// Mitsubishi GX Works2 project: hello   PLC: Q03UDV

PROGRAM MAIN
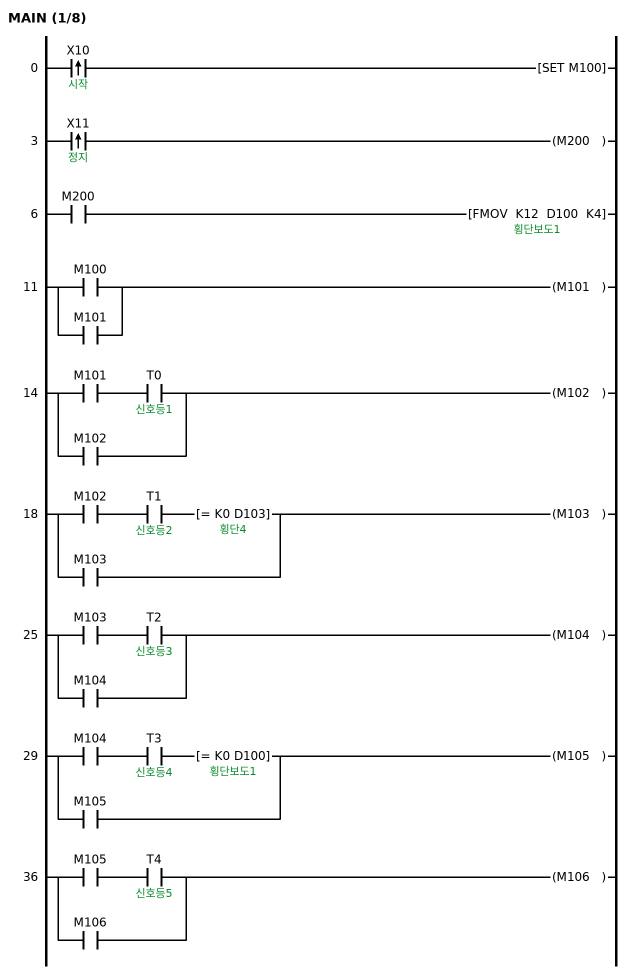
0     LDP     X10  ; 시작
      SET     M100
3     LDP     X11  ; 정지
      OUT     M200
6     LD      M200
      FMOV    K12 D100 K4  ; 횡단보도1
11    LD      M100
      OR      M101
      OUT     M101
14    LD      M101
      AND     T0  ; 신호등1
      OR      M102
      OUT     M102
18    LD      M102
      AND     T1  ; 신호등2
      AND=    K0 D103  ; 횡단4
      OR      M103
      OUT     M103
25    LD      M103
      AND     T2  ; 신호등3
      OR      M104
      OUT     M104
29    LD      M104
      AND     T3  ; 신호등4
      AND=    K0 D100  ; 횡단보도1
      OR      M105
      OUT     M105
36    LD      M105
      AND     T4  ; 신호등5
      OR      M106
      OUT     M106
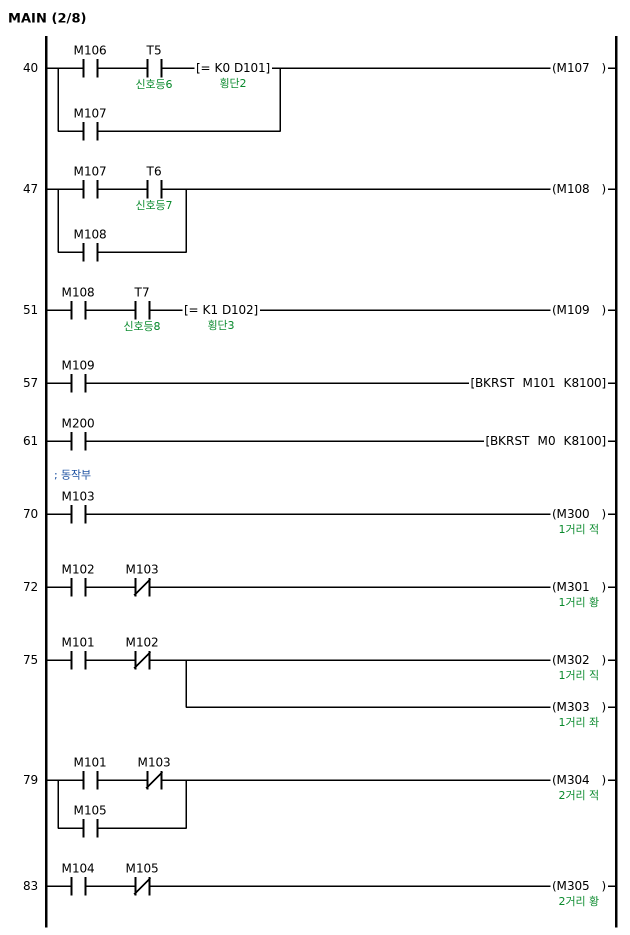
40    LD      M106
      AND     T5  ; 신호등6
      AND=    K0 D101  ; 횡단2
      OR      M107
      OUT     M107
47    LD      M107
      AND     T6  ; 신호등7
      OR      M108
      OUT     M108
51    LD      M108
      AND     T7  ; 신호등8
      AND=    K1 D102  ; 횡단3
      OUT     M109
57    LD      M109
      BKRST   M101 K8100
61    LD      M200
      BKRST   M0 K8100
; 동작부
70    LD      M103
      OUT     M300  ; 1거리 적
72    LD      M102
      ANI     M103
      OUT     M301  ; 1거리 황
75    LD      M101
      ANI     M102
      OUT     M302  ; 1거리 직
      OUT     M303  ; 1거리 좌
79    LD      M101
      ANI     M103
      OR      M105
      OUT     M304  ; 2거리 적
83    LD      M104
      ANI     M105
      OUT     M305  ; 2거리 황
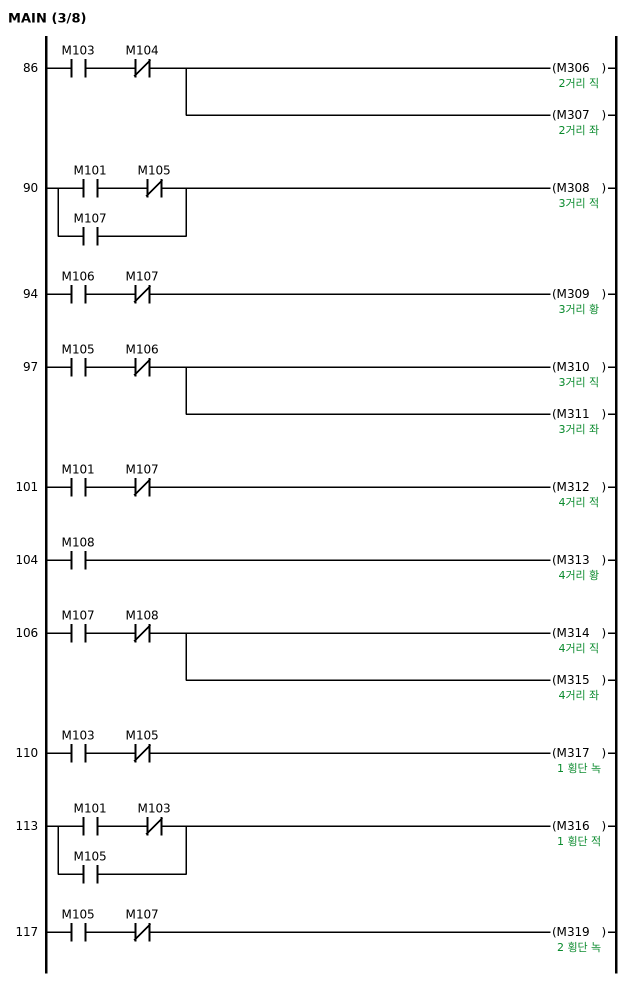
86    LD      M103
      ANI     M104
      OUT     M306  ; 2거리 직
      OUT     M307  ; 2거리 좌
90    LD      M101
      ANI     M105
      OR      M107
      OUT     M308  ; 3거리 적
94    LD      M106
      ANI     M107
      OUT     M309  ; 3거리 황
97    LD      M105
      ANI     M106
      OUT     M310  ; 3거리 직
      OUT     M311  ; 3거리 좌
101   LD      M101
      ANI     M107
      OUT     M312  ; 4거리 적
104   LD      M108
      OUT     M313  ; 4거리 황
106   LD      M107
      ANI     M108
      OUT     M314  ; 4거리 직
      OUT     M315  ; 4거리 좌
110   LD      M103
      ANI     M105
      OUT     M317  ; 1 횡단 녹
113   LD      M101
      ANI     M103
      OR      M105
      OUT     M316  ; 1 횡단 적
117   LD      M105
      ANI     M107
      OUT     M319  ; 2 횡단 녹
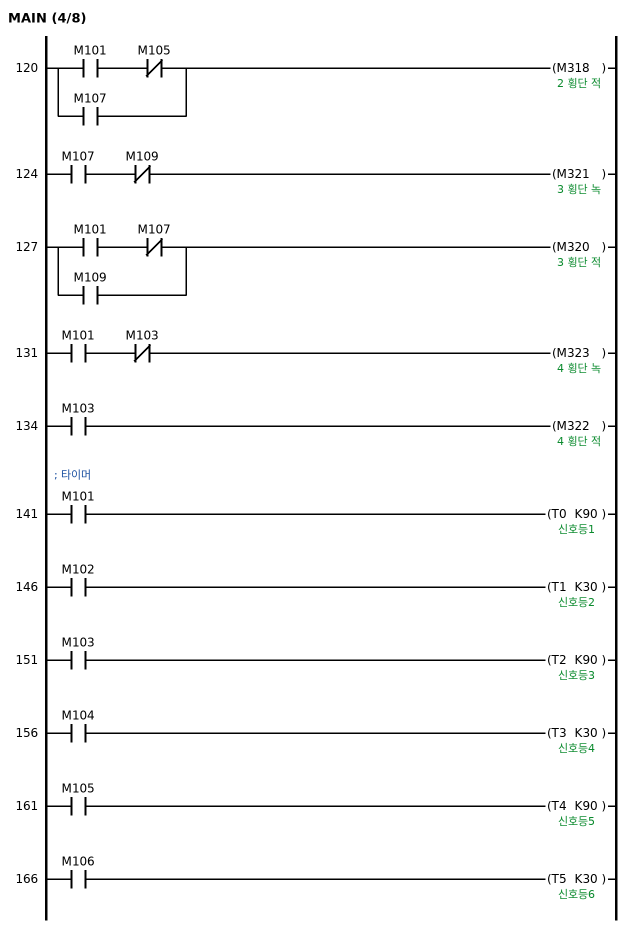
120   LD      M101
      ANI     M105
      OR      M107
      OUT     M318  ; 2 횡단 적
124   LD      M107
      ANI     M109
      OUT     M321  ; 3 횡단 녹
127   LD      M101
      ANI     M107
      OR      M109
      OUT     M320  ; 3 횡단 적
131   LD      M101
      ANI     M103
      OUT     M323  ; 4 횡단 녹
134   LD      M103
      OUT     M322  ; 4 횡단 적
; 타이머
141   LD      M101
      OUT     T0 K90  ; 신호등1
146   LD      M102
      OUT     T1 K30  ; 신호등2
151   LD      M103
      OUT     T2 K90  ; 신호등3
156   LD      M104
      OUT     T3 K30  ; 신호등4
161   LD      M105
      OUT     T4 K90  ; 신호등5
166   LD      M106
      OUT     T5 K30  ; 신호등6
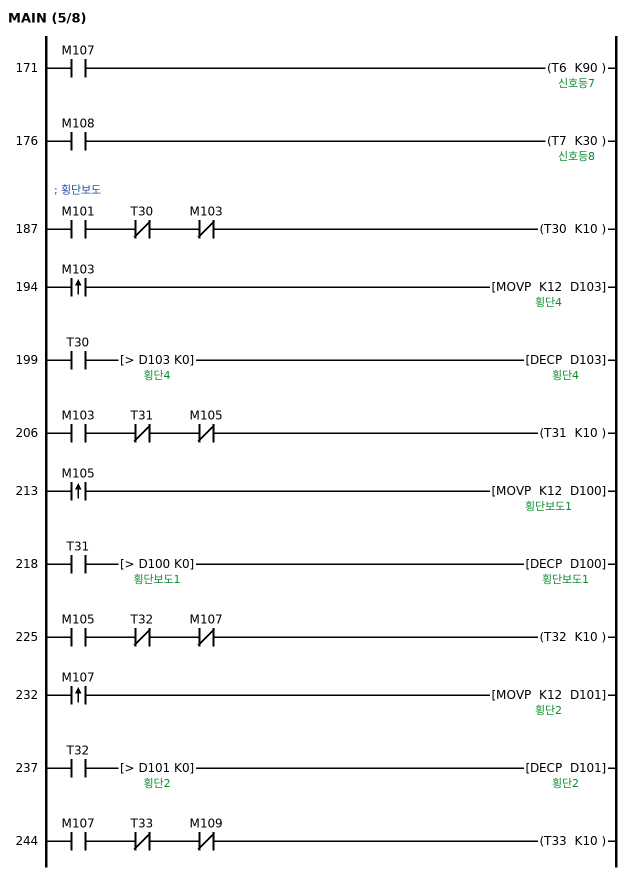
171   LD      M107
      OUT     T6 K90  ; 신호등7
176   LD      M108
      OUT     T7 K30  ; 신호등8
; 횡단보도
187   LD      M101
      ANI     T30
      ANI     M103
      OUT     T30 K10
194   LDP     M103
      MOVP    K12 D103
199   LD      T30
      AND>    D103 K0  ; 횡단4
      DECP    D103
206   LD      M103
      ANI     T31
      ANI     M105
      OUT     T31 K10
213   LDP     M105
      MOVP    K12 D100
218   LD      T31
      AND>    D100 K0  ; 횡단보도1
      DECP    D100
225   LD      M105
      ANI     T32
      ANI     M107
      OUT     T32 K10
232   LDP     M107
      MOVP    K12 D101
237   LD      T32
      AND>    D101 K0  ; 횡단2
      DECP    D101
244   LD      M107
      ANI     T33
      ANI     M109
      OUT     T33 K10
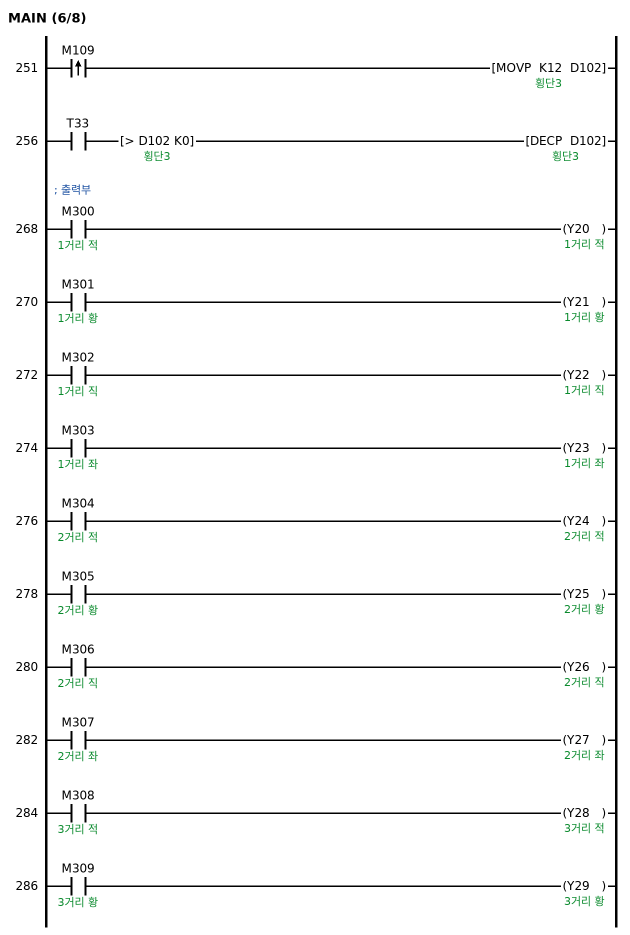
251   LDP     M109
      MOVP    K12 D102
256   LD      T33
      AND>    D102 K0  ; 횡단3
      DECP    D102
; 출력부
268   LD      M300  ; 1거리 적
      OUT     Y20  ; 1거리 적
270   LD      M301  ; 1거리 황
      OUT     Y21  ; 1거리 황
272   LD      M302  ; 1거리 직
      OUT     Y22  ; 1거리 직
274   LD      M303  ; 1거리 좌
      OUT     Y23  ; 1거리 좌
276   LD      M304  ; 2거리 적
      OUT     Y24  ; 2거리 적
278   LD      M305  ; 2거리 황
      OUT     Y25  ; 2거리 황
280   LD      M306  ; 2거리 직
      OUT     Y26  ; 2거리 직
282   LD      M307  ; 2거리 좌
      OUT     Y27  ; 2거리 좌
284   LD      M308  ; 3거리 적
      OUT     Y28  ; 3거리 적
286   LD      M309  ; 3거리 황
      OUT     Y29  ; 3거리 황
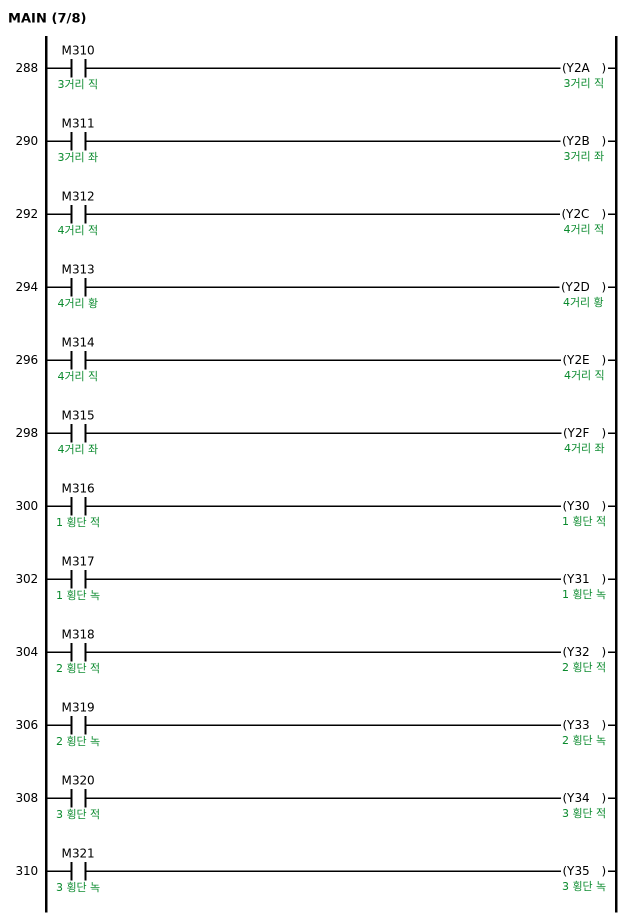
288   LD      M310  ; 3거리 직
      OUT     Y2A  ; 3거리 직
290   LD      M311  ; 3거리 좌
      OUT     Y2B  ; 3거리 좌
292   LD      M312  ; 4거리 적
      OUT     Y2C  ; 4거리 적
294   LD      M313  ; 4거리 황
      OUT     Y2D  ; 4거리 황
296   LD      M314  ; 4거리 직
      OUT     Y2E  ; 4거리 직
298   LD      M315  ; 4거리 좌
      OUT     Y2F  ; 4거리 좌
300   LD      M316  ; 1 횡단 적
      OUT     Y30  ; 1 횡단 적
302   LD      M317  ; 1 횡단 녹
      OUT     Y31  ; 1 횡단 녹
304   LD      M318  ; 2 횡단 적
      OUT     Y32  ; 2 횡단 적
306   LD      M319  ; 2 횡단 녹
      OUT     Y33  ; 2 횡단 녹
308   LD      M320  ; 3 횡단 적
      OUT     Y34  ; 3 횡단 적
310   LD      M321  ; 3 횡단 녹
      OUT     Y35  ; 3 횡단 녹
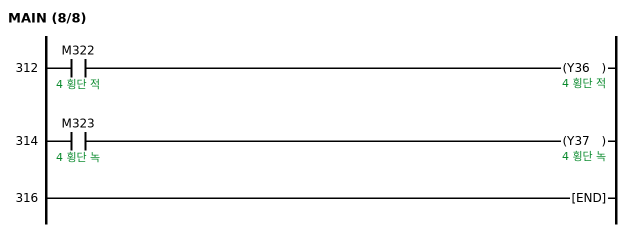
312   LD      M322  ; 4 횡단 적
      OUT     Y36  ; 4 횡단 적
314   LD      M323  ; 4 횡단 녹
      OUT     Y37  ; 4 횡단 녹
316   END
END_PROGRAM

PROGRAM upgrade
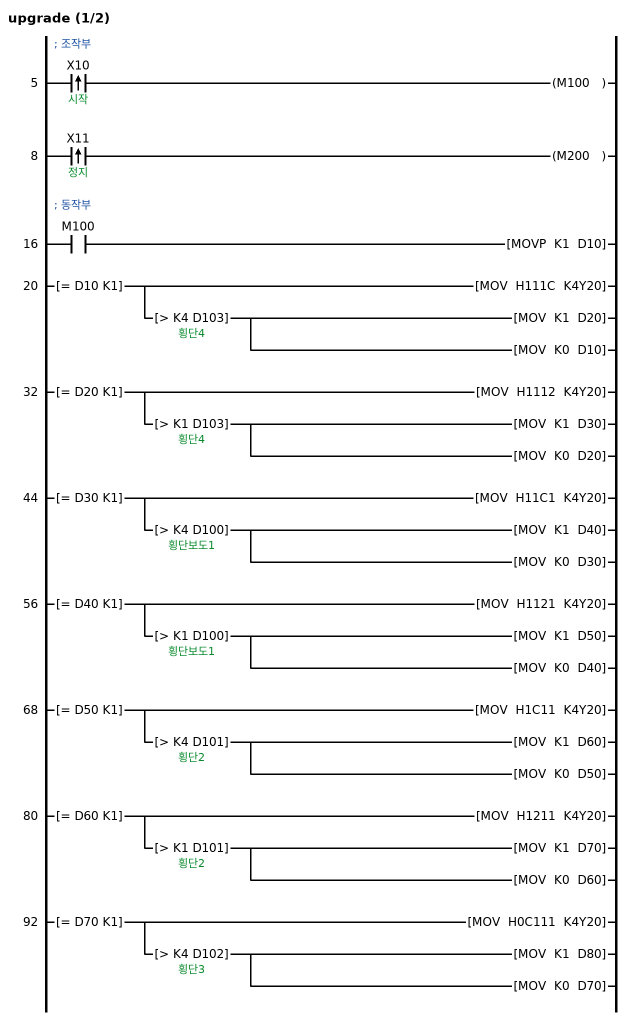
; 조작부
5     LDP     X10  ; 시작
      OUT     M100
8     LDP     X11  ; 정지
      OUT     M200
; 동작부
16    LD      M100
      MOVP    K1 D10
20    LD=     D10 K1
      MOV     H111C K4Y20  ; 1거리 적
      AND>    K4 D103  ; 횡단4
      MOV     K1 D20
      MOV     K0 D10
32    LD=     D20 K1
      MOV     H1112 K4Y20
      AND>    K1 D103  ; 횡단4
      MOV     K1 D30
      MOV     K0 D20
44    LD=     D30 K1
      MOV     H11C1 K4Y20
      AND>    K4 D100  ; 횡단보도1
      MOV     K1 D40
      MOV     K0 D30
56    LD=     D40 K1
      MOV     H1121 K4Y20
      AND>    K1 D100  ; 횡단보도1
      MOV     K1 D50
      MOV     K0 D40
68    LD=     D50 K1
      MOV     H1C11 K4Y20
      AND>    K4 D101  ; 횡단2
      MOV     K1 D60
      MOV     K0 D50
80    LD=     D60 K1
      MOV     H1211 K4Y20
      AND>    K1 D101  ; 횡단2
      MOV     K1 D70
      MOV     K0 D60
92    LD=     D70 K1
      MOV     H0C111 K4Y20
      AND>    K4 D102  ; 횡단3
      MOV     K1 D80
      MOV     K0 D70
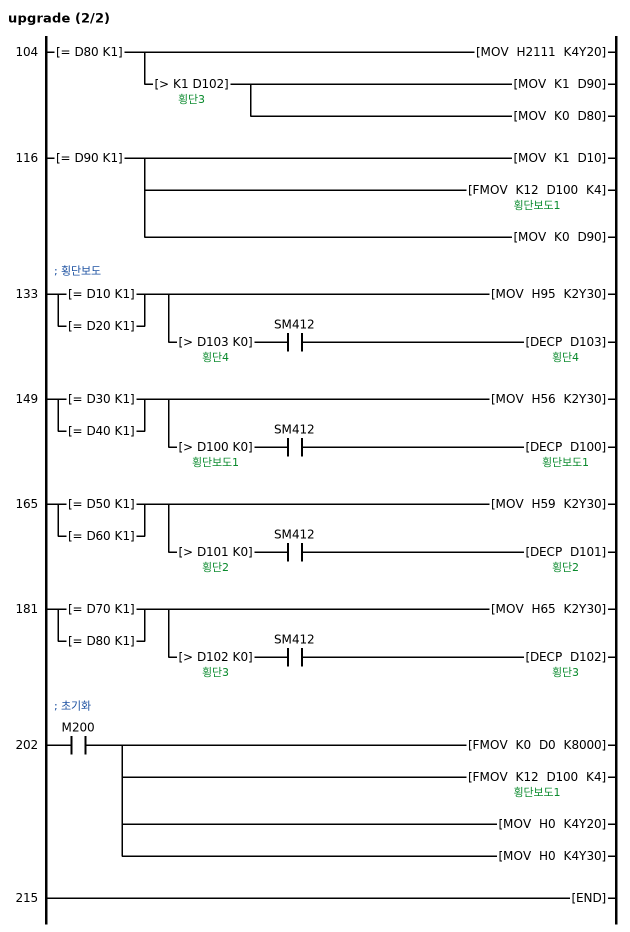
104   LD=     D80 K1
      MOV     H2111 K4Y20
      AND>    K1 D102  ; 횡단3
      MOV     K1 D90
      MOV     K0 D80
116   LD=     D90 K1
      MOV     K1 D10
      FMOV    K12 D100 K4
      MOV     K0 D90
; 횡단보도
133   LD=     D10 K1
      OR=     D20 K1
      MOV     H95 K2Y30  ; 1 횡단 적
      AND>    D103 K0  ; 횡단4
      AND     SM412
      DECP    D103
149   LD=     D30 K1
      OR=     D40 K1
      MOV     H56 K2Y30
      AND>    D100 K0  ; 횡단보도1
      AND     SM412
      DECP    D100
165   LD=     D50 K1
      OR=     D60 K1
      MOV     H59 K2Y30
      AND>    D101 K0  ; 횡단2
      AND     SM412
      DECP    D101
181   LD=     D70 K1
      OR=     D80 K1
      MOV     H65 K2Y30
      AND>    D102 K0  ; 횡단3
      AND     SM412
      DECP    D102
; 초기화
202   LD      M200
      FMOV    K0 D0 K8000
      FMOV    K12 D100 K4
      MOV     H0 K4Y20
      MOV     H0 K4Y30
215   END
END_PROGRAM

PROGRAM nowait
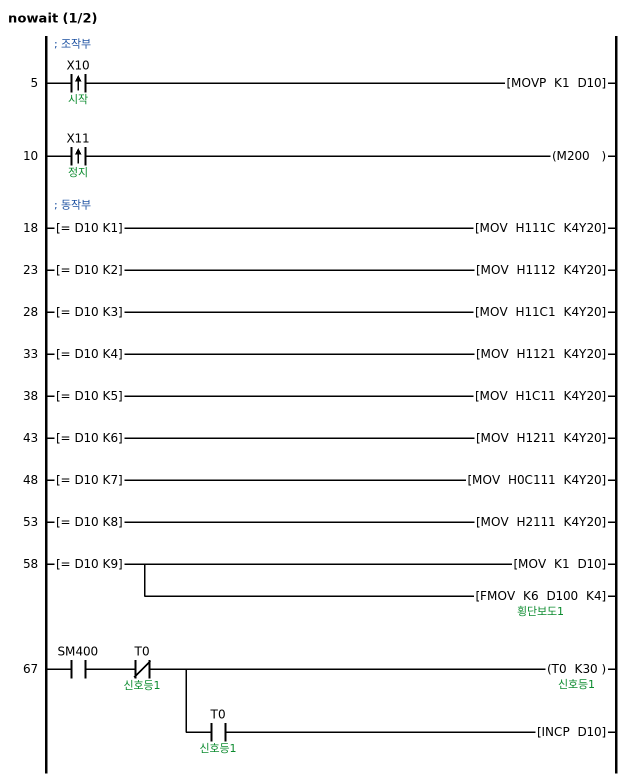
; 조작부
5     LDP     X10  ; 시작
      MOVP    K1 D10
10    LDP     X11  ; 정지
      OUT     M200
; 동작부
18    LD=     D10 K1
      MOV     H111C K4Y20  ; 1거리 적
23    LD=     D10 K2
      MOV     H1112 K4Y20
28    LD=     D10 K3
      MOV     H11C1 K4Y20
33    LD=     D10 K4
      MOV     H1121 K4Y20
38    LD=     D10 K5
      MOV     H1C11 K4Y20
43    LD=     D10 K6
      MOV     H1211 K4Y20
48    LD=     D10 K7
      MOV     H0C111 K4Y20
53    LD=     D10 K8
      MOV     H2111 K4Y20
58    LD=     D10 K9
      MOV     K1 D10
      FMOV    K6 D100 K4  ; 횡단보도1
67    LD      SM400
      ANI     T0  ; 신호등1
      OUT     T0 K30  ; 신호등1
      AND     T0  ; 신호등1
      INCP    D10
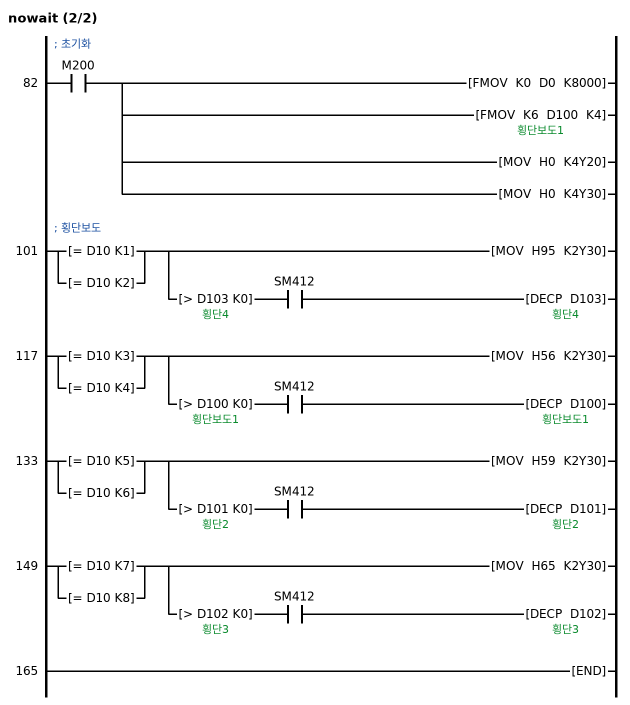
; 초기화
82    LD      M200
      FMOV    K0 D0 K8000
      FMOV    K6 D100 K4
      MOV     H0 K4Y20
      MOV     H0 K4Y30  ; 1 횡단 적
; 횡단보도
101   LD=     D10 K1
      OR=     D10 K2
      MOV     H95 K2Y30
      AND>    D103 K0  ; 횡단4
      AND     SM412
      DECP    D103
117   LD=     D10 K3
      OR=     D10 K4
      MOV     H56 K2Y30
      AND>    D100 K0  ; 횡단보도1
      AND     SM412
      DECP    D100
133   LD=     D10 K5
      OR=     D10 K6
      MOV     H59 K2Y30
      AND>    D101 K0  ; 횡단2
      AND     SM412
      DECP    D101
149   LD=     D10 K7
      OR=     D10 K8
      MOV     H65 K2Y30
      AND>    D102 K0  ; 횡단3
      AND     SM412
      DECP    D102
165   END
END_PROGRAM

PROGRAM Watch
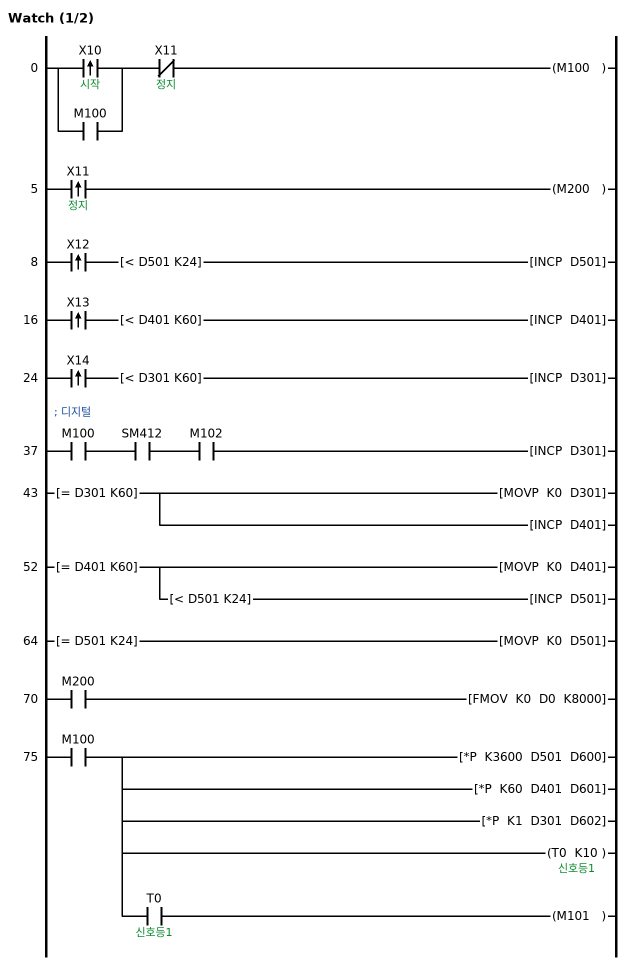
0     LDP     X10  ; 시작
      OR      M100
      ANI     X11  ; 정지
      OUT     M100
5     LDP     X11  ; 정지
      OUT     M200
8     LDP     X12
      AND<    D501 K24
      INCP    D501
16    LDP     X13
      AND<    D401 K60
      INCP    D401
24    LDP     X14
      AND<    D301 K60
      INCP    D301
; 디지털
37    LD      M100
      AND     SM412
      AND     M102
      INCP    D301
43    LD=     D301 K60
      MOVP    K0 D301
      INCP    D401
52    LD=     D401 K60
      MOVP    K0 D401
      AND<    D501 K24
      INCP    D501
64    LD=     D501 K24
      MOVP    K0 D501
70    LD      M200
      FMOV    K0 D0 K8000
75    LD      M100
      *P      K3600 D501 D600
      *P      K60 D401 D601
      *P      K1 D301 D602
      OUT     T0 K10  ; 신호등1
      AND     T0  ; 신호등1
      OUT     M101
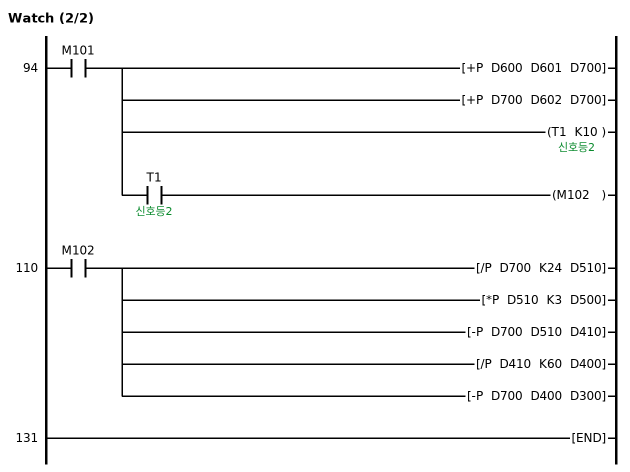
94    LD      M101
      +P      D600 D601 D700
      +P      D700 D602 D700
      OUT     T1 K10  ; 신호등2
      AND     T1  ; 신호등2
      OUT     M102
110   LD      M102
      /P      D700 K24 D510
      *P      D510 K3 D500
      -P      D700 D510 D410
      /P      D410 K60 D400
      -P      D700 D400 D300
131   END
END_PROGRAM
